Universal Robots PolyScope program: orange_Hospital_small_top.urp

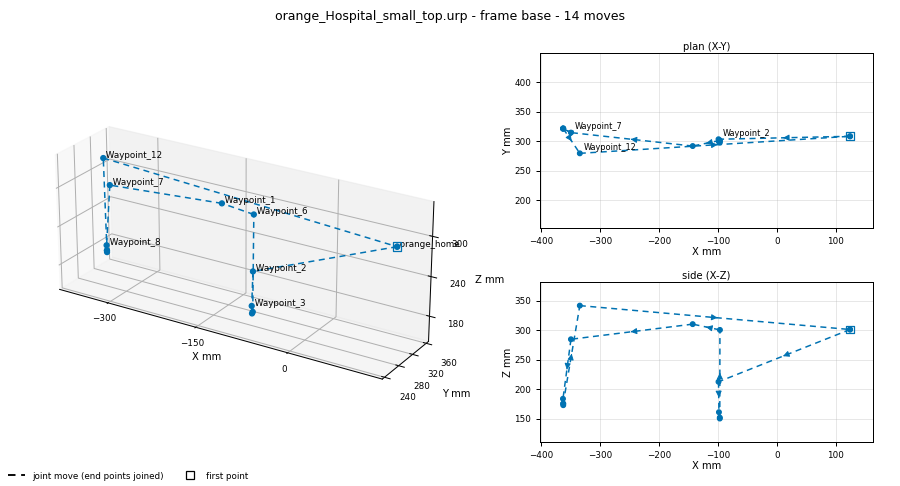
[picture p0: tool path of orange_Hospital_small_top.urp in frame base, 14 of 14 moves have a stored position in this frame; points joined in program order, loops and branches not executed]
Program orange_Hospital_small_top (installation=default directory=/programs/usbdisk/Zahra1/orangi createdIn=5.11.11.1010533 lastSavedIn=5.11.11.1010533 robotSerialNumber=20205300864)
Calibrated DH parameters: a=[-0.000166, -0.243494, -0.153108, 0.000057, -0.000123, 0]; d=[0.151897, -1.34267, 53.988124, -52.514559, 0.085283, 0.092193]; alpha=[1.572472, -0.003756, 0.002824, 1.570807, -1.572621, 0]; deltaTheta=[0, 0.020704, 7.033215, -0.770746, 0.000004, 0]
Robot Program (runOnlyOnce=true)
  MoveJ speed 60 deg/s, acceleration 80 deg/s^2 (useActiveTCP=true) feature=Base
    Waypoint orange_home: TCP in base x=124.286 y=308.277 z=301.462 mm, rx=2.2499 ry=-2.1846 rz=-0.0963 rad; joints [-269.66, -91.226, -90.279, -86.086, 92.69, 808.818] deg
    URCap Gripper (Robotiq_Grippers, Robotiq Inc.) dataModel(position=41.96078431372549, force=70.0, speed=18.0, positionInDouble=41.96078431372549, forceInDouble=70.0, speedInDouble=18.0, slaveIds=[9], blocking=true, robotCompliant=false)
    Waypoint Waypoint_2: TCP in base x=-98.975 y=303.254 z=212.759 mm, rx=2.1816 ry=-2.189 rz=-0.0391 rad; joints [-228.774, -93.173, -112.508, -62.945, 93.05, 851.624] deg
    Waypoint Waypoint_3: TCP in base x=-98.255 y=299.022 z=161.117 mm, rx=2.2053 ry=-2.205 rz=-0.0367 rad; joints [-227.824, -99.414, -121.977, -47.216, 91.401, 852.392] deg
    Waypoint Waypoint_4: TCP in base x=-96.811 y=297.564 z=150.351 mm, rx=2.183 ry=-2.2103 rz=-0.0345 rad; joints [-228.065, -101.168, -123.642, -43.901, 92.076, 852.885] deg
    URCap Gripper (Robotiq_Grippers, Robotiq Inc.) dataModel(position=72.54901960784314, force=46.0, speed=18.0, positionInDouble=72.54901960784314, forceInDouble=46.0, speedInDouble=18.0, slaveIds=[9], blocking=true, robotCompliant=true)
    Waypoint Waypoint_5: motionParameters(jointSpeed=0.698132 jointAcceleration=0.349066 cartesianSpeed=0.25 cartesianAcceleration=1.2); TCP in base x=-96.808 y=299.469 z=151.995 mm, rx=2.1802 ry=-2.2117 rz=-0.0341 rad; joints [-228.338, -101.251, -122.902, -44.581, 92.134, 852.724] deg
    Waypoint Waypoint_6: TCP in base x=-96.584 y=301.283 z=300.801 mm, rx=2.1907 ry=-2.2181 rz=-0.0122 rad; joints [-228.327, -87.624, -93.216, -88.675, 91.431, 852.497] deg
    Waypoint Waypoint_1: TCP in base x=-142.804 y=291.711 z=310.569 mm, rx=2.2888 ry=-2.1095 rz=-0.1681 rad; joints [-220.605, -87.656, -93.039, -82.968, 91.195, 854.9] deg
    Waypoint Waypoint_7: TCP in base x=-349.477 y=314.552 z=284.896 mm, rx=0.0126 ry=-3.0259 rz=-0.1038 rad; joints [-205.721, -125.619, -50.3, -86.393, 89.213, 963.797] deg
    Waypoint Waypoint_8: TCP in base x=-363.029 y=321.432 z=183.855 mm, rx=-0.0555 ry=-3.1338 rz=-0.0126 rad; joints [-205.875, -135.204, -57.868, -76.251, 89.65, 966.223] deg
    Waypoint Waypoint_9: TCP in base x=-362.602 y=321.385 z=175.612 mm, rx=0.0549 ry=3.1329 rz=0.0065 rad; joints [-205.862, -135.926, -58.449, -75.845, 89.48, 966.221] deg
    Waypoint Waypoint_10: motionParameters(jointSpeed=0.698132 jointAcceleration=0.349066 cartesianSpeed=0.25 cartesianAcceleration=1.2); TCP in base x=-362.562 y=321.403 z=172.994 mm, rx=0.0549 ry=3.1329 rz=0.0065 rad; joints [-205.866, -136.104, -58.844, -75.275, 89.478, 966.215] deg
    URCap Gripper (Robotiq_Grippers, Robotiq Inc.) dataModel(position=31.764705882352942, force=50.0, speed=18.0, positionInDouble=31.764705882352942, forceInDouble=50.0, speedInDouble=18.0, slaveIds=[9], blocking=true, robotCompliant=true)
    Waypoint Waypoint_9: TCP in base x=-362.602 y=321.385 z=175.612 mm, rx=0.0549 ry=3.1329 rz=0.0065 rad; joints [-205.862, -135.926, -58.449, -75.845, 89.48, 966.221] deg
    Waypoint Waypoint_12: TCP in base x=-334.427 y=279.344 z=342.03 mm, rx=-0.0692 ry=-3.0677 rz=-0.1164 rad; joints [-201.819, -118.451, -45.266, -100.848, 87.243, 970.676] deg
    Waypoint orange_home: TCP in base x=124.286 y=308.277 z=301.462 mm, rx=2.2499 ry=-2.1846 rz=-0.0963 rad; joints [-269.66, -91.226, -90.279, -86.086, 92.69, 808.818] deg
